// TIA Portal V18 export
// export: Created 2026-06-08T16:52:55.8113714Z, ExportSetting WithDefaults, DisplayName Totally Integrated Automation Portal, DisplayVersion V18, DisplayName TIA Portal Openness, DisplayVersion V18, DisplayName TIA Portal Version Control Interface, DisplayVersion V18, DisplayName STEP 7 Professional, DisplayVersion V18, DisplayName STEP 7 Safety, DisplayVersion V18, DisplayName WinCC Professional, DisplayVersion V18
ORGANIZATION_BLOCK "Main"   // OB1, LAD, ProgramCycle
TITLE = "Main Program Sweep (Cycle)"
{ S7_Optimized_Access := 'TRUE' }
VERSION : 0.1
// stored: AutoNumber true, IsIECCheckEnabled false, SetENOAutomatically false
   VAR_INPUT
      Initial_Call : Bool;   // Initial call of this OB
      Remanence : Bool;   // =True, if remanent data are available
   END_VAR
   VAR_TEMP   // added for the SCL form of the ladder/FBD networks
      _w1 : Bool;
   END_VAR
BEGIN

REGION Network 1
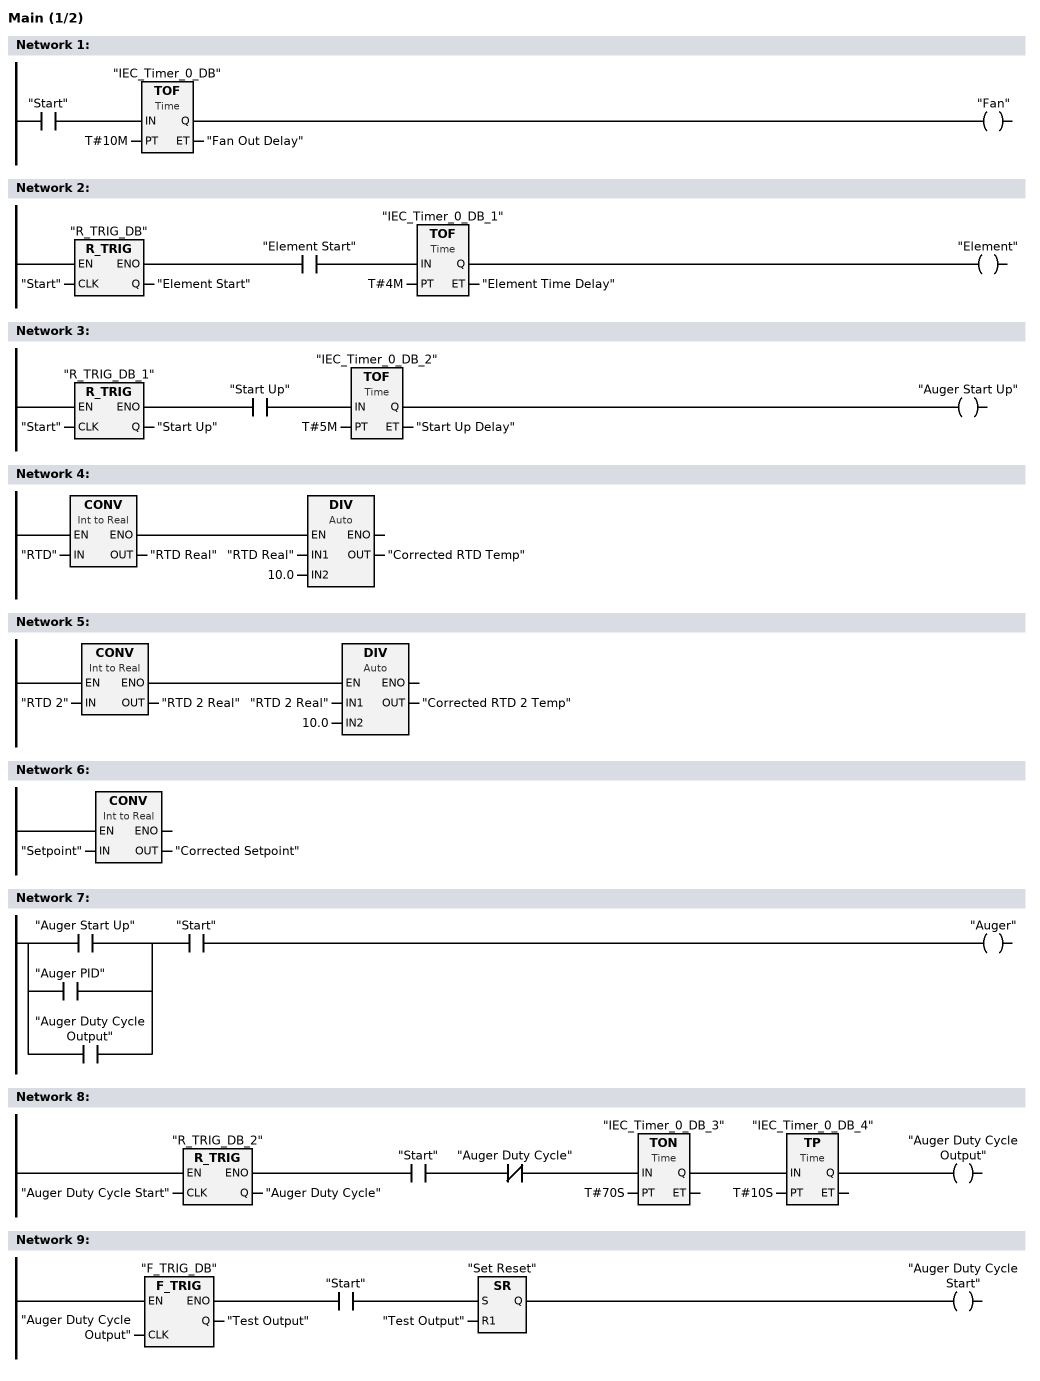
   RUNG wire#powerrail
      Contact( "Start" )
      { S7_Templates := "time_type := Time" } "IEC_Timer_0_DB".TOF(pt := T#10M, et => "Fan Out Delay")
      Coil( "Fan" )
   END_RUNG
   // the same network as SCL:
   "IEC_Timer_0_DB".TOF(IN := "Start", PT := T#10M, ET => "Fan Out Delay");
   "Fan" := "IEC_Timer_0_DB".Q;
END_REGION

REGION Network 2
   RUNG wire#powerrail
      "R_TRIG_DB".R_TRIG(CLK := "Start", Q => "Element Start")
      Contact( "Element Start" )
      { S7_Templates := "time_type := Time" } "IEC_Timer_0_DB_1".TOF(pt := T#4M, et => "Element Time Delay")
      Coil( "Element" )
   END_RUNG
   // the same network as SCL:
   "R_TRIG_DB"(CLK := "Start", Q => "Element Start", ENO => #_w1);   // R_TRIG
   "IEC_Timer_0_DB_1".TOF(IN := #_w1 AND "Element Start", PT := T#4M, ET => "Element Time Delay");
   "Element" := "IEC_Timer_0_DB_1".Q;
END_REGION

REGION Network 3
   RUNG wire#powerrail
      "R_TRIG_DB_1".R_TRIG(CLK := "Start", Q => "Start Up")
      Contact( "Start Up" )
      { S7_Templates := "time_type := Time" } "IEC_Timer_0_DB_2".TOF(pt := T#5M, et => "Start Up Delay")
      Coil( "Auger Start Up" )
   END_RUNG
   // the same network as SCL:
   "R_TRIG_DB_1"(CLK := "Start", Q => "Start Up", ENO => #_w1);   // R_TRIG
   "IEC_Timer_0_DB_2".TOF(IN := #_w1 AND "Start Up", PT := T#5M, ET => "Start Up Delay");
   "Auger Start Up" := "IEC_Timer_0_DB_2".Q;
END_REGION

REGION Network 4
   RUNG wire#powerrail
      { S7_Templates := "[SrcType := Int, DestType := Real]" } Convert(in := "RTD", out => "RTD Real")
      Div(in1 := "RTD Real", in2 := 10.0, out => "Corrected RTD Temp")
   END_RUNG
   // the same network as SCL:
   "RTD Real" := INT_TO_REAL("RTD");
   "Corrected RTD Temp" := "RTD Real" / 10.0;
END_REGION

REGION Network 5
   RUNG wire#powerrail
      { S7_Templates := "[SrcType := Int, DestType := Real]" } Convert(in := "RTD 2", out => "RTD 2 Real")
      Div(in1 := "RTD 2 Real", in2 := 10.0, out => "Corrected RTD 2 Temp")
   END_RUNG
   // the same network as SCL:
   "RTD 2 Real" := INT_TO_REAL("RTD 2");
   "Corrected RTD 2 Temp" := "RTD 2 Real" / 10.0;
END_REGION

REGION Network 6
   RUNG wire#powerrail
      { S7_Templates := "[SrcType := Int, DestType := Real]" } Convert(in := "Setpoint", out => "Corrected Setpoint")
   END_RUNG
   // the same network as SCL:
   "Corrected Setpoint" := INT_TO_REAL("Setpoint");
END_REGION

REGION Network 7
   RUNG wire#powerrail
      Contact( "Auger Start Up" )
      wire#w1
      Contact( "Start" )
      Coil( "Auger" )
   END_RUNG
   RUNG wire#powerrail
      Contact( "Auger PID" )
   END_RUNG wire#w1
   RUNG wire#powerrail
      Contact( "Auger Duty Cycle Output" )
   END_RUNG wire#w1
   // the same network as SCL:
   "Auger" := ("Auger Start Up" OR "Auger PID" OR "Auger Duty Cycle Output") AND "Start";
END_REGION

REGION Network 8
   RUNG wire#powerrail
      "R_TRIG_DB_2".R_TRIG(CLK := "Auger Duty Cycle Start", Q => "Auger Duty Cycle")
      Contact( "Start" )
      I_Contact( "Auger Duty Cycle" )
      { S7_Templates := "time_type := Time" } "IEC_Timer_0_DB_3".TON(pt := T#70S, et =>)
      { S7_Templates := "time_type := Time" } "IEC_Timer_0_DB_4".TP(pt := T#10S, et =>)
      Coil( "Auger Duty Cycle Output" )
   END_RUNG
   // the same network as SCL:
   "R_TRIG_DB_2"(CLK := "Auger Duty Cycle Start", Q => "Auger Duty Cycle", ENO => #_w1);   // R_TRIG
   "IEC_Timer_0_DB_3".TON(IN := #_w1 AND "Start" AND NOT "Auger Duty Cycle", PT := T#70S);
   "IEC_Timer_0_DB_4".TP(IN := "IEC_Timer_0_DB_3".Q, PT := T#10S);
   "Auger Duty Cycle Output" := "IEC_Timer_0_DB_4".Q;
END_REGION

REGION Network 9
   RUNG wire#powerrail
      "F_TRIG_DB".F_TRIG(CLK := "Auger Duty Cycle Output", Q => "Test Output")
      Contact( "Start" )
      S_SR(operand := "Set Reset", r1 := "Test Output")
      Coil( "Auger Duty Cycle Start" )
   END_RUNG
   // the same network as SCL:
   "F_TRIG_DB"(CLK := "Auger Duty Cycle Output", Q => "Test Output", ENO => #_w1);   // F_TRIG
   IF #_w1 AND "Start" THEN
       "Set Reset" := TRUE;   // SR flip-flop
   END_IF;
   IF "Test Output" THEN "Set Reset" := FALSE; END_IF;
   "Auger Duty Cycle Start" := "Set Reset";
END_REGION

REGION Network 10
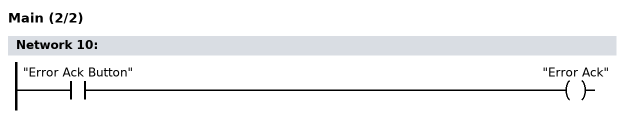
   RUNG wire#powerrail
      Contact( "Error Ack Button" )
      Coil( "Error Ack" )
   END_RUNG
   // the same network as SCL:
   "Error Ack" := "Error Ack Button";
END_REGION
END_ORGANIZATION_BLOCK
